TYPE ST_Robot_Mitsubishi_Packet_2013 :
STRUCT
	// Packet number - 2013.
	// To robot.
	// Robot stop control packet.
	// Trigger.
	
	Header							: DINT := 2013;													// Packet header.

END_STRUCT
END_TYPE

(* stored: Version 1.1.0.1, ProductVersion 3.1.4024.3
   DUT ST_Robot_Mitsubishi_Packet_2013: Id {77f99491-9a33-4904-9371-d7a2966b19b7} *)
